// TIA Portal V17 export
// export: Created 2022-07-20T06:59:49.566329Z, ExportSetting WithDefaults, DisplayName Totally Integrated Automation Portal, DisplayVersion V17, DisplayName TIA Portal Openness, DisplayVersion V17, DisplayName TIA Portal Version Control Interface, DisplayVersion V17, DisplayName SINAMICS Startdrive Advanced, DisplayVersion V17, DisplayName SINAMICS Startdrive G130, G150, S120, S150, SINAMICS MV, S210, DisplayVersion V17, DisplayName SINAMICS Startdrive G110M, G120, G120C, G120D, G120P, G115D, DisplayVersion V17, DisplayName STEP 7 Professional, DisplayVersion V17, DisplayName STEP 7 Safety, DisplayVersion V17, DisplayName WinCC Advanced, DisplayVersion V17
FUNCTION "FC10022_DoubleTolerenceRelation" : Void   // FC10022, LAD
{ S7_Optimized_Access := 'TRUE' }
VERSION : 0.1
// stored: AutoNumber false, IsIECCheckEnabled false, SetENOAutomatically false, UDAEnableTagReadback false
   VAR_INPUT
      ActualPositionMaster : Real;
      ActualPositionSlave : Real;
      PositionTested : Real;
      Tolerance : Real;
   END_VAR
   VAR_OUTPUT
      InPosition : Bool;
   END_VAR
   VAR_TEMP
      MasterInPos : Bool;
      SlaveInPos : Bool;
   END_VAR
BEGIN

REGION Network 1 (SCL)
   IF ((#PositionTested - #Tolerance) <= #ActualPositionMaster) AND ((#PositionTested + #Tolerance) >= #ActualPositionMaster) THEN
       #MasterInPos := true;
   ELSE
       #MasterInPos := false;
   END_IF;

   IF ((#PositionTested - #Tolerance) <= #ActualPositionSlave) AND ((#PositionTested + #Tolerance) >= #ActualPositionSlave) THEN
       #SlaveInPos := true;
   ELSE
       #SlaveInPos := false;
   END_IF;

   #InPosition := #MasterInPos AND #SlaveInPos;
END_REGION
END_FUNCTION
